(* PLC project Unnamed, Unknown Unnamed 1 *)
(* stored: creationDateTime 2026-07-15T10:53:28, modificationDateTime 2026-07-15T10:53:28 *)

FUNCTION DIV : ANY_NUM
  VAR_INPUT
    IN1 : ANY_NUM;
    IN2 : ANY_NUM;
  END_VAR

END_FUNCTION

FUNCTION MOVE : ANY
  VAR_INPUT
    IN : ANY;
  END_VAR

END_FUNCTION

FUNCTION SUB : ANY_NUM
  VAR_INPUT
    IN1 : ANY_NUM;
    IN2 : ANY_NUM;
  END_VAR

END_FUNCTION

PROGRAM main
  VAR
    PC_ANPR_Truk_Detected AT %QX0.0 : BOOL;
    S1_LiDAR_Posisi AT %QX0.1 : BOOL;
    S2_LoadCell_Stable AT %QX0.2 : BOOL;
    Reset_Button AT %QX0.3 : BOOL;
    Palang_masuk AT %QX0.4 : BOOL;
    Sistem_Ready AT %QX0.5 : BOOL;
    Alarm_Posisi AT %QX0.6 : BOOL;
    Lock_Data AT %QX0.7 : BOOL;
    LiDAR_Volume_Raw AT %QW1 : UINT;
    LoadCell_Weight_Raw AT %QW2 : UINT;
    Database_Tare_Weight AT %QW3 : UINT;
    Netto_Weight AT %QW4 : UINT;
    Density_Result AT %QW5 : UINT;
  END_VAR
  VAR
    Volume_Locked : UINT;
    Weight_Locked : UINT;
  END_VAR

(* LD diagram, written out as Structured Text *)
Palang_masuk := NOT Lock_Data AND PC_ANPR_Truk_Detected;
Sistem_Ready := NOT Lock_Data;
Alarm_Posisi := PC_ANPR_Truk_Detected AND NOT S1_LiDAR_Posisi;
Lock_Data := (Lock_Data OR PC_ANPR_Truk_Detected AND S1_LiDAR_Posisi AND S2_LoadCell_Stable) AND NOT Reset_Button;
IF Lock_Data THEN Volume_Locked := LiDAR_Volume_Raw; END_IF;
IF Lock_Data THEN Weight_Locked := LoadCell_Weight_Raw; END_IF;
IF Lock_Data THEN Netto_Weight := Weight_Locked - Database_Tare_Weight; END_IF;
IF Lock_Data THEN Density_Result := Netto_Weight / Volume_Locked; END_IF;
END_PROGRAM

CONFIGURATION Config0
  RESOURCE Res0 ON PLC
    TASK task0(INTERVAL := T#20ms, PRIORITY := 1);
    PROGRAM instance0 WITH task0 : main;
  END_RESOURCE
END_CONFIGURATION
